ABB RobotStudio station: 手爪更换1.0.rsstn

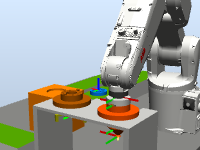
Station Station (saved by RobotStudio 6.4.7206.1027)
Controller System1, task T_ROB1: task frame (RAPID world) sits at (0, -189.91, 800) mm in the station
Controller System1
  mechanical unit ROB_1: IRB1200_5_90_STD_02, 6 joints, base frame (0, 0, 0) mm
Layout (positions relative to the parent item):
  - IRB1200_5_90_STD_02 [mechanism, from Robots\IRB1200_5_90_STD_02.rslib] at (0, -189.91, 800) mm; joint values [1.7401, 0.8984, -0.2519, 0, 0.9243, 1.7401] (rad or m)
  - 装配台 [part]
  - 部件 [part] at (-223.98, -561.16, 0) mm
  - 部件_2 [part] at (0, -203.49, 0) mm
  - 部件_3 [part] at (-693.25, 1032.81, 0) mm
  - 部件_4 [part] at (1137.19, 901.79, 0) mm, rotated rx 0 ry 0 rz -90 deg
  - 部件_5 [part] at (943.53, 901.79, 0) mm, rotated rx 0 ry 0 rz -90 deg
  - 零件1 [part] at (456.45, -184.74, 900.36) mm
  - 零件2 [part] at (649, -852.3, 901.96) mm
  - 工具母头组件 [smart component] at (-123.98, 535.34, 1158) mm, rotated rx 180 ry 0 rz 180 deg
      signals: DI qijin
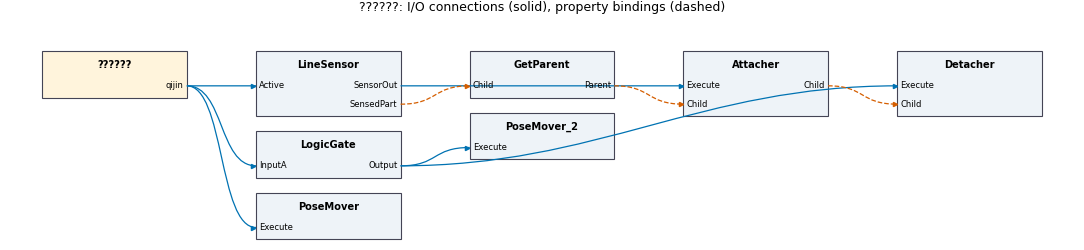
      connections:
        工具母头组件.qijin -> LineSensor.Active
        LineSensor.SensorOut -> Attacher.Execute
        工具母头组件.qijin -> LogicGate.InputA
        LogicGate.Output -> Detacher.Execute
        工具母头组件.qijin -> PoseMover.Execute
        LogicGate.Output -> PoseMover_2.Execute
        Attacher.Child => Detacher.Child
        LineSensor.SensedPart => GetParent.Child
        GetParent.Parent => Attacher.Child
    - 工具母头 [mechanism] at (600, 0, 1100.94) mm, rotated rx 180 ry 0 rz 180 deg; joint values [0, 0] (rad or m)
        TCP changtool at (0, 0, -20) mm
        TCP xipan at (0, 0, -140) mm
        TCP jiazhua at (0, 0, -106) mm
        links: L1, L2, L3
    - Attacher [smart component, from Components\Attacher.rslib] at (600, 0, 1100.94) mm, rotated rx 180 ry 0 rz 180 deg
        properties: Parent=工具母头; Flange=0; Child=吸盘组件; Mount=false; Offset=[0 0 0]; Orientation=[0 0 0]
    - Detacher [smart component, from Components\Detacher.rslib] at (600, 0, 1100.94) mm, rotated rx 180 ry 0 rz 180 deg
        properties: Child=吸盘组件; KeepPosition=true
    - LineSensor [smart component, from Components\LineSensor.rslib] at (600, 0, 1100.94) mm, rotated rx 180 ry 0 rz 180 deg
        properties: Start=[0.6 0 1.07794]; End=[0.6 0 1.03794]; Radius=0.002; SensedPart=吸盘; SensedPoint=[-0.123978004455566 0.535344970703125 1.108]
      - _sensorPart_ [part]
    - LogicGate [smart component, from Components\LogicGate.rslib] at (600, 0, 1100.94) mm, rotated rx 180 ry 0 rz 180 deg
        properties: Operator=NOT; Delay=0
    - PoseMover [smart component, from Components\PoseMover.rslib] at (600, 0, 1100.94) mm, rotated rx 180 ry 0 rz 180 deg
        properties: Mechanism=工具母头; Pose=2; Duration=0
    - PoseMover_2 [smart component, from Components\PoseMover.rslib] at (600, 0, 1100.94) mm, rotated rx 180 ry 0 rz 180 deg
        properties: Mechanism=工具母头; Pose=0; Duration=0
    - GetParent [smart component, from Components\GetParent.rslib]
        properties: Child=吸盘; Parent=吸盘组件
  - 吸盘 [graphiccomponentgroup]
  - 爪子组件 [smart component]
      signals: DI zhuazi
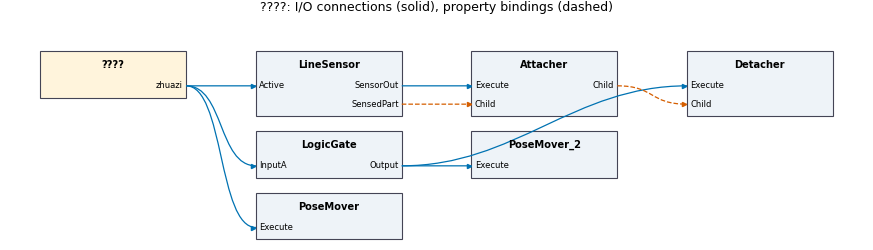
      connections:
        爪子组件.zhuazi -> LineSensor.Active
        LineSensor.SensorOut -> Attacher.Execute
        爪子组件.zhuazi -> LogicGate.InputA
        LogicGate.Output -> Detacher.Execute
        爪子组件.zhuazi -> PoseMover.Execute
        LogicGate.Output -> PoseMover_2.Execute
        LineSensor.SensedPart => Attacher.Child
        Attacher.Child => Detacher.Child
    - 爪子 [mechanism] at (-523.98, 535.35, 59.15) mm; joint values [0.025, 0.025, 0.025] (rad or m)
        links: L1, L2, L3, L4
    - LogicGate [smart component, from Components\LogicGate.rslib]
        properties: Operator=NOT; Delay=0
    - LineSensor [smart component, from Components\LineSensor.rslib]
        properties: Start=[0.07602 0.53535 1.065]; End=[0.07602 0.53535 1.043]; Radius=0.002; SensedPart=(none); SensedPoint=[0 0 0]
      - _sensorPart_ [part]
    - Attacher [smart component, from Components\Attacher.rslib]
        properties: Parent=工具母头组件; Flange=0; Child=(none); Mount=false; Offset=[0 0 0]; Orientation=[0 0 0]
    - Detacher [smart component, from Components\Detacher.rslib]
        properties: Child=(none); KeepPosition=true
    - PoseMover [smart component, from Components\PoseMover.rslib]
        properties: Mechanism=爪子; Pose=2; Duration=0.5
    - PoseMover_2 [smart component, from Components\PoseMover.rslib]
        properties: Mechanism=爪子; Pose=0; Duration=0.5
    - maitoulinjian [part] at (0, 0, -40.83) mm
  - 吸盘组件 [smart component]
      signals: DI xipan
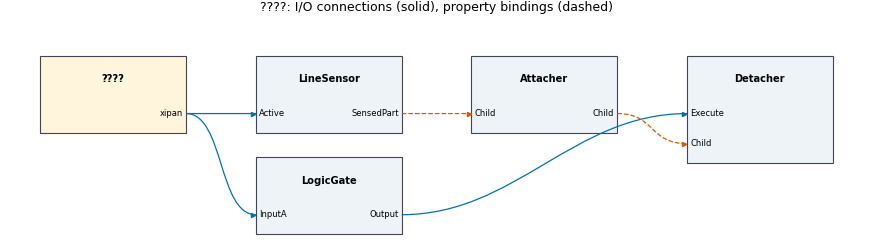
      connections:
        吸盘组件.xipan -> LineSensor.Active
        吸盘组件.xipan -> LogicGate.InputA
        LogicGate.Output -> Detacher.Execute
        LineSensor.SensedPart => Attacher.Child
        Attacher.Child => Detacher.Child
    - LineSensor [smart component, from Components\LineSensor.rslib]
        properties: Start=[-0.123978 0.535345 1.016]; End=[-0.123978 0.535345 1.003]; Radius=0.002; SensedPart=(none); SensedPoint=[0 0 0]
      - _sensorPart_ [part]
    - LogicGate [smart component, from Components\LogicGate.rslib]
        properties: Operator=NOT; Delay=0
    - Attacher [smart component, from Components\Attacher.rslib]
        properties: Parent=吸盘组件; Flange=0; Child=(none); Mount=false; Offset=[0 0 0]; Orientation=[0 0 0]
    - Detacher [smart component, from Components\Detacher.rslib]
        properties: Child=(none); KeepPosition=true
    - 吸盘 [part] at (-123.98, 535.34, 788.76) mm
Attachment: 工具母头组件 is attached to IRB1200_5_90_STD_02 / Link6
Targets, tools, work objects and paths stored in the station, written as RAPID:
! task T_ROB1
MODULE CalibData
  PERS tooldata changtool:=[TRUE,[[0,0,19.999],[0,0,1,0]],[1,[-1,0,0],[1,0,0,0],0,0,0]];
  PERS tooldata xipan:=[TRUE,[[0,0,140],[0,0,1,0]],[1,[-1,0,0],[1,0,0,0],0,0,0]];
  PERS tooldata jiazhua:=[TRUE,[[0,0,105.999],[0,0,1,0]],[1,[-1,0,0],[1,0,0,0],0,0,0]];
ENDMODULE

! task T_ROB1
MODULE Module1
  CONST robtarget tool2change:=[[-123.978,725.255,251.999],[1,0,0,0],[0,0,0,0],[9E+09,9E+09,9E+09,9E+09,9E+09,9E+09]];
  CONST robtarget tool1change:=[[76.02,725.26,254.422112025],[1,0,0,0],[0,0,0,0],[9E+09,9E+09,9E+09,9E+09,9E+09,9E+09]];
  CONST robtarget xiaolan:=[[456.446,5.167,120.36],[1,0,0,0],[0,0,0,0],[9E+09,9E+09,9E+09,9E+09,9E+09,9E+09]];
ENDMODULE

